FUNCTION_BLOCK FB_GeoPosition_Test EXTENDS FB_TestSuite
VAR_INPUT
END_VAR
VAR_OUTPUT
END_VAR
VAR
END_VAR

WhenValuesSetExpectValuesRetained();

METHOD PRIVATE WhenValuesSetExpectValuesRetained
VAR_INPUT
	
END_VAR
VAR
	P1 : GeoPosition;
	P1b : GeoPosition;
	P2 : GeoPosition;
	P3 : GeoPosition;
END_VAR
TEST('WhenValuesSetExpectValuesRetained');

// @TEST-RUN
P1.SetFromComponentsRad(PI,PI,1);
P1b.SetFromComponentsRad(PI,PI,1);
P2 := P1;
P3.SetFromComponentsDeg(180,180,1);

// @TEST-ASSERT
AssertTrue(P1.IsEqual(P1b), 'equals check does not work');
AssertTrue(P1.IsEqual(P3),'radians and degrees do not agree');
AssertTrue(P2.LatitudeDeg > 179.99,'latitude not retained');
AssertTrue(P2.LongitudeDeg > 179.99,'longitude not retained');
AssertTrue(P2.Elevation = 1,'elevation not retained');


TEST_FINISHED();
END_METHOD

END_FUNCTION_BLOCK

(* stored: Version 1.1.0.1, ProductVersion 3.1.4024.9
   POU FB_GeoPosition_Test: Id {9c8846f8-6574-4c98-87c7-35162f85ac9e}, SpecialFunc None
   Method WhenValuesSetExpectValuesRetained: Id {2d895917-8468-4b71-bf91-ddd149f04fe2} *)
